PROGRAM pouMachine
VAR
	pnuOn: FB_Motion1way;
	isAirSwitchOn: BOOL;
END_VAR
VAR // added by the converter: edge detectors and wires of the graphical bodies
    _w1 : BOOL;
END_VAR

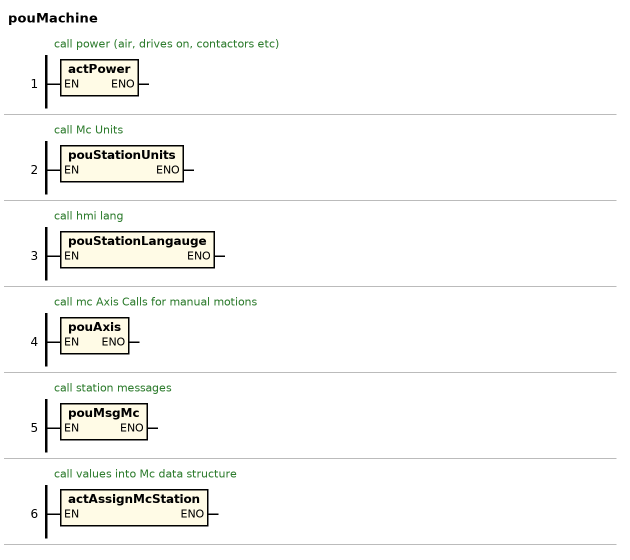
// NETWORK 1
// call power (air, drives on, contactors etc)
actPower();

// NETWORK 2
// call Mc Units
pouStationUnits();

// NETWORK 3
// call hmi lang
pouStationLangauge();

// NETWORK 4
// call mc Axis Calls for manual motions
pouAxis();

// NETWORK 5
// call station messages
pouMsgMc();

// NETWORK 6
// call values into Mc data structure
actAssignMcStation();

ACTION actAssignMcStation:
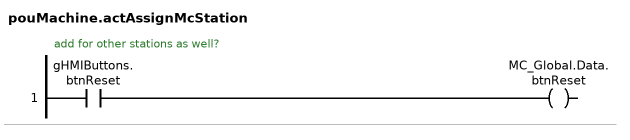
// NETWORK 1
// add for other stations as well?
MC_Global.Data.btnReset := gHMIButtons.btnReset;
END_ACTION

ACTION actPower:
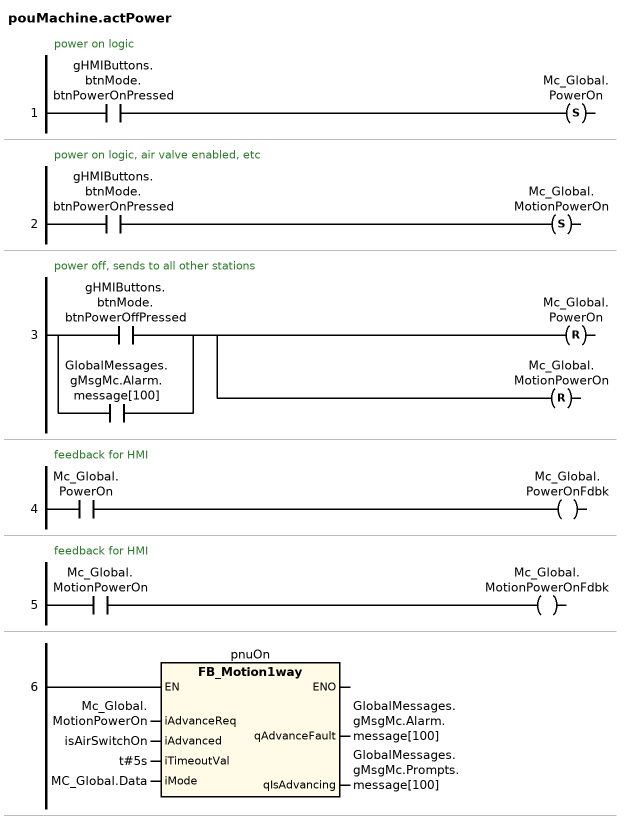
// NETWORK 1
// power on logic
Mc_Global.PowerOn S= gHMIButtons.btnMode.btnPowerOnPressed;

// NETWORK 2
// power on logic, air valve enabled, etc
Mc_Global.MotionPowerOn S= gHMIButtons.btnMode.btnPowerOnPressed;

// NETWORK 3
// power off, sends to all other stations
_w1 := gHMIButtons.btnMode.btnPowerOffPressed OR GlobalMessages.gMsgMc.Alarm.message[100];
Mc_Global.PowerOn R= _w1;
Mc_Global.MotionPowerOn R= _w1;

// NETWORK 4
// feedback for HMI
Mc_Global.PowerOnFdbk := Mc_Global.PowerOn;

// NETWORK 5
// feedback for HMI
Mc_Global.MotionPowerOnFdbk := Mc_Global.MotionPowerOn;

// NETWORK 6
pnuOn(
    iAdvanceReq := Mc_Global.MotionPowerOn,
    iAdvanced := isAirSwitchOn,
    iTimeoutVal := t#5s,
    iMode := MC_Global.Data,
    qAdvanceFault => GlobalMessages.gMsgMc.Alarm.message[100],
    qIsAdvancing => GlobalMessages.gMsgMc.Prompts.message[100]); // FB_Motion1way
END_ACTION

END_PROGRAM

(* stored: Version 1.1.0.1, ProductVersion 3.1.4024.12
   POU pouMachine: Id {130f38d3-d0ad-451a-83e5-25f291f23105}, SpecialFunc None
   Action actAssignMcStation: Id {86f27bdf-cbff-4efe-a514-d6c2d712b080}
   Action actPower: Id {2ab649fa-87ba-4e15-a599-af17da8737b9} *)
